ABB RobotStudio station: Solution1_20190225-114000.rsstn

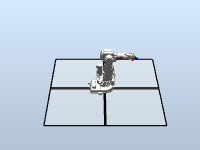
Station Solution1 (saved by RobotStudio 6.8.8148.134)
Controller IRB_140_6kg_0.81m
  mechanical unit ROB_1: IRB140_6_81_C_03_2, 6 joints, base frame (0, 0, 0) mm
Layout (positions relative to the parent item):
  - IRB140_6_81_C_03 [mechanism, from Robots\IRB140_6_81_C_G_03.rslib] at (0, 0, 0) mm; joint values [0, 0, 0, 0, 0.5236, 0] (rad or m)
  - IRB140_6_81_C_03_2 [mechanism, from Robots\IRB140_6_81_C_G_03.rslib] at (0, 0, 0) mm; joint values [0, 0, 0, 0, 0.5236, 0] (rad or m)
Targets, tools, work objects and paths stored in the station, written as RAPID:
! task T_ROB1
MODULE Module1
  PROC main()
    MoveL pHOME,v1000,fine,tool0;
    MoveL p10,v1000,fine,tool0;
    MoveL pHOME,v1000,fine,tool0;
  ENDPROC
ENDMODULE

! task T_ROB1
MODULE Module1
  PROC Path_10()
  ENDPROC
ENDMODULE

